FUNCTION_BLOCK FB_Module_ToolHolderDoor IMPLEMENTS I_Module
VAR_INPUT
	sName			: STRING[50];
	tTimeout		: TIME := T#0S;
END_VAR

VAR_IN_OUT
END_VAR

VAR_OUTPUT
	bEnabled     	: BOOL;
	eState			: E_State := E_State.DISABLED;
	eNextState		: E_State := E_State.DISABLED;
	sStatusText 	: STRING[100];
	
	bDoorOpening	: BOOL;
	bDoorClosing	: BOOL;
END_VAR

VAR
	eLastState		: E_State;
	tTimeoutTimer	: TON;
	Components		: ARRAY [0..0] OF I_Component;	
	fbPiston		: FB_Component_DualValveGuarded;
END_VAR

VAR CONSTANT
	DISABLED		: E_State := E_State.DISABLED;
	READY			: E_State := E_State.READY;
	BUSY			: E_State := E_State.BUSY;
	HALTED			: E_State := E_State.HALTED;
	TIMEOUT			: E_State := E_State.TIMEOUT;
END_VAR

tTimeoutTimer(PT := tTimeout);

fbPiston(	sName 			:= 'piston for toolholder door', 
			bSensExtended 	:= GVL.bDoorToolHolderDown, 
			bSensRetracted 	:= GVL.bDoorToolHolderLock, 
			bOutputA 		:= GVL.bOpenToolCarrierDoor, 
			bOutputB 		:= GVL.bCloseToolCarrierDoor); 
			
Components[0] := fbPiston;

eState := eNextState;

CASE eState OF
	DISABLED: 	sStatusText := 'tool holder door is disabled';
	READY: 		sStatusText := 'tool holder door is ready to operate';
	BUSY: 		IF bDoorOpening THEN
					sStatusText := 'door opening';
					IF fbPiston.bIsExtended THEN
						bDoorOpening 	:= FALSE;
						eNextState 		:= TIMEOUT;
					END_IF
				ELSIF bDoorClosing THEN
					sStatusText := 'door closing';
					IF fbPiston.bIsRetracted THEN
						bDoorClosing 	:= FALSE;
						eNextState 		:= TIMEOUT;
					END_IF
				END_IF
				
	TIMEOUT:	sStatusText := 'Tool holder door is in timeout';
				tTimeoutTimer(IN := TRUE);
				
				IF tTimeoutTimer.Q THEN
					tTimeoutTimer(IN := FALSE);
					eNextState := READY;
				END_IF
				
	HALTED:		sStatusText := 'Tool holder door is halted';
END_CASE

METHOD M_Close : BOOL
VAR_INPUT
END_VAR
IF eState = READY OR eState = BUSY THEN
	eNextState 		:= BUSY;
	bDoorClosing 	:= TRUE;
	fbPiston.M_Retract();
END_IF
END_METHOD

{warning 'add method implementation '}
METHOD M_Disable : BOOL

VAR
	idx: INT;
END_VAR
IF eState = READY THEN
	bEnabled	:= FALSE;
	eNextState	:= DISABLED;
	
	FOR idx := 0 TO 0 DO
    	Components[idx].M_Disable();
	END_FOR;
END_IF
END_METHOD

{warning 'add method implementation '}
METHOD M_Enable : BOOL

VAR
	idx: INT;
END_VAR
IF eState = DISABLED THEN
	bEnabled	:= TRUE;
	eNextState	:= READY;
	
	FOR idx := 0 TO 0 DO
    	Components[idx].M_Enable();
	END_FOR;
END_IF
END_METHOD

{warning 'add method implementation '}
METHOD M_Halt : BOOL

VAR
	idx: INT;
END_VAR
IF eState <> HALTED AND eState <> DISABLED THEN
	eLastState 		:= eState;
	eNextState		:= HALTED;
	FOR idx := 0 TO 0 DO
		Components[idx].M_Halt();
	END_FOR;
END_IF
END_METHOD

METHOD M_Open : BOOL
VAR_INPUT
END_VAR
IF eState = READY OR eState = BUSY THEN
	eNextState 		:= BUSY;
	bDoorOpening 	:= TRUE;
	fbPiston.M_Extend();
END_IF
END_METHOD

{warning 'add method implementation '}
METHOD M_Resume : BOOL

VAR
	idx: INT;
END_VAR
IF eState = HALTED THEN
	eNextState := eLastState;
	FOR idx := 0 TO 0 DO
		Components[idx].M_Resume();
	END_FOR;
END_IF
END_METHOD

END_FUNCTION_BLOCK

(* stored: Version 1.1.0.1, ProductVersion 3.1.4024.15
   POU FB_Module_ToolHolderDoor: Id {f6e0d382-5b3d-4622-b685-26d7f0ea4bef}, SpecialFunc None
   Method M_Close: Id {9e689a25-9200-4c78-98dc-720336982544}
   Method M_Disable: Id {94b3cc84-0f56-40ff-85e0-e7d35b21966a}
   Method M_Enable: Id {9c1b8958-2725-46b8-9769-57cd4e6b810e}
   Method M_Halt: Id {8e27d0bc-9254-4f5a-b07b-532e2d31a0bc}
   Method M_Open: Id {f29e878a-65dd-40bb-b2c6-4ae134b78d2b}
   Method M_Resume: Id {0500d455-1511-46bd-a4db-9fb0599c6e7c} *)
